FUNCTION BoolToErrorText : STRING
VAR_INPUT
	Error: BOOL;
END_VAR
VAR
END_VAR

IF Error THEN
	BoolToErrorText := 'Error';
ELSE
	BoolToErrorText := 'OK';
END_IF

END_FUNCTION

(* stored: Version 1.1.0.1, ProductVersion 3.1.4024.6
   POU BoolToErrorText: Id {1c47d453-b9a0-4fef-acb9-dc5b5c2621ca}, SpecialFunc None *)
